{attribute 'linkalways'} 
{attribute 'no_explicit_call' := 'This FB is a CLASS and must be accessed using methods or properties'}
{attribute 'enable_dynamic_creation'}
FUNCTION_BLOCK _ETcVnCodeDetectionModel EXTENDS EnumDatatypeBase
VAR
	localData : ETcVnCodeDetectionModel;
	activeData : REFERENCE TO ETcVnCodeDetectionModel;
	enumBaseDatatype : _ULINT(localData);
END_VAR

METHOD PRIVATE AddLocalEnumeration
VAR_INPUT
	Enumeration : T_MAXSTRING;
	Value : ETcVnCodeDetectionModel;
END_VAR
AddEnumeration(Enumeration, Value);
END_METHOD

PROPERTY PUBLIC Address : PVOID
GET
Address := ADR(activeData);
END_GET
END_PROPERTY

METHOD PUBLIC ClearReference
VAR_INPUT
END_VAR
activeData REF= localData;
SetBaseDatatypeReference();
END_METHOD

METHOD PUBLIC Clone : I_Datatype
VAR
    pClone : POINTER TO _ETcVnCodeDetectionModel;
END_VAR
pClone := __NEW(_ETcVnCodeDetectionModel(InitialValue := Value));
Clone := pClone^;
END_METHOD

METHOD FB_init : BOOL
VAR_INPUT
	bInitRetains : BOOL; // if TRUE, the retain variables are initialized (warm start / cold start)
	bInCopyCode : BOOL;  // if TRUE, the instance afterwards gets moved into the copy code (online change)
	InitialValue : ETcVnCodeDetectionModel;
END_VAR
localData := InitialValue;
AddBaseDatatype(enumBaseDatatype);
ClearReference();

AddLocalEnumeration('TCVN_CDM_DETECT_1_1', ETcVnCodeDetectionModel.TCVN_CDM_DETECT_1_1);
AddLocalEnumeration('TCVN_CDM_DETECT_1_2', ETcVnCodeDetectionModel.TCVN_CDM_DETECT_1_2);
AddLocalEnumeration('TCVN_CDM_DETECT_1_3', ETcVnCodeDetectionModel.TCVN_CDM_DETECT_1_3);
AddLocalEnumeration('TCVN_CDM_DETECT_2_1', ETcVnCodeDetectionModel.TCVN_CDM_DETECT_2_1);
AddLocalEnumeration('TCVN_CDM_DETECT_2_2', ETcVnCodeDetectionModel.TCVN_CDM_DETECT_2_2);
AddLocalEnumeration('TCVN_CDM_DETECT_2_3', ETcVnCodeDetectionModel.TCVN_CDM_DETECT_2_3);
AddLocalEnumeration('TCVN_CDM_DETECT_3_1', ETcVnCodeDetectionModel.TCVN_CDM_DETECT_3_1);
AddLocalEnumeration('TCVN_CDM_DETECT_3_2', ETcVnCodeDetectionModel.TCVN_CDM_DETECT_3_2);
AddLocalEnumeration('TCVN_CDM_DETECT_3_3', ETcVnCodeDetectionModel.TCVN_CDM_DETECT_3_3);
END_METHOD

PROPERTY PUBLIC Identifier : T_MAXSTRING
GET
Identifier := 'ETcVnCodeDetectionModel';
END_GET
END_PROPERTY

METHOD IsEnumeratorValueEqual : BOOL
VAR_INPUT
	Enumerator : I_KeyValueForwardEnumerator;
END_VAR
VAR
	storedValue : ETcVnCodeDetectionModel;
END_VAR
IF NOT Enumerator.TryGet(storedValue) THEN
	RETURN;
END_IF

IsEnumeratorValueEqual := storedValue = activeData;
END_METHOD

METHOD PUBLIC MakeReferenceTo
VAR_INPUT
	ReferenceTarget : REFERENCE TO ETcVnCodeDetectionModel;
END_VAR
activeData REF= ReferenceTarget;
SetBaseDatatypeReference();
END_METHOD

METHOD PROTECTED SetBaseDatatypeReference
VAR_INPUT
END_VAR
enumBaseDatatype.MakeReferenceTo(activeData);
END_METHOD

PROPERTY PUBLIC Size : UDINT
GET
Size := SIZEOF(activeData);
END_GET
END_PROPERTY

METHOD TryMakeReferenceTo : BOOL
VAR_INPUT
	Target : I_Datatype;
END_VAR
VAR
	pTargetData : POINTER TO ETcVnCodeDetectionModel;
END_VAR
IF NOT IsEquivalentTo(Target) THEN
	RETURN;
END_IF

pTargetData := Target.Address;
activeData REF= pTargetData^;
SetBaseDatatypeReference();
TryMakeReferenceTo := TRUE;
END_METHOD

PROPERTY PUBLIC Value : ETcVnCodeDetectionModel
GET
Value := activeData;
END_GET
SET
activeData := Value;
END_SET
END_PROPERTY

END_FUNCTION_BLOCK

(* stored: Version 1.1.0.1, ProductVersion 3.1.4026.13
   POU _ETcVnCodeDetectionModel: Id {bb0b3d12-6c29-0e8c-2e85-938d608e62b1}, SpecialFunc None
   Folder Core: Id {6faceb99-ebfe-053e-3e25-a5c00f3583c1}
   Folder Protected: Id {ea8f3f8a-aebe-0fbd-1bc3-690a8a426a26}
   Folder Customize: Id {8e3998be-5cce-0fca-13f0-b14cd0f4ce24}
   Folder Constructor: Id {1fed5bcb-d668-0785-0360-4cd6b93e187b}
   Folder Private: Id {caac75eb-2f55-0d0d-248d-78e3be7f8da4}
   Folder Protected: Id {ea2d5394-47bd-0485-3c81-24915d245fcf}
   Method AddLocalEnumeration: Id {fe58a232-2f00-0a52-18d1-8e5afb100686}
   Property Address: Id {6ab8040c-d31b-0e81-2098-9c6e21e3f357}
   Get Get: Id {61c1a01e-6d2a-065a-29da-cd9581289d3f}
   Method ClearReference: Id {78abd788-dbf9-08b7-0fbc-bb4212861b25}
   Method Clone: Id {b6bced59-98bd-0a89-2fa8-15db095ae1cc}
   Method FB_init: Id {4b3cc9dd-10e0-0f24-3e56-a36e90fdd84a}
   Property Identifier: Id {1fe61a0e-c48f-0101-3461-084250fb6792}
   Get Get: Id {ab4c16b6-7cc2-0662-3318-83d8195380aa}
   Method IsEnumeratorValueEqual: Id {13272841-da9f-08aa-2cb9-efffc2b437ef}
   Method MakeReferenceTo: Id {dbc33961-663e-05d0-1533-1d1fb076c605}
   Method SetBaseDatatypeReference: Id {c1fa98da-d7c8-022f-2cf9-c9b99ff5fecd}
   Property Size: Id {8ef02a02-512e-04b9-3dd1-9284dd9e246f}
   Get Get: Id {82f552c2-d9cc-0299-0616-8621d82261f2}
   Method TryMakeReferenceTo: Id {7a78c074-9f58-047f-1c0a-cf2edea0279b}
   Property Value: Id {8e4d9b55-a9fd-0254-123d-f457419aa976}
   Get Get: Id {d33cb1be-e390-0337-23ff-903e70b1fb7d}
   Set Set: Id {266ec089-29ba-0882-304a-a6f4d232ab21} *)
